FUNCTION_BLOCK FB_StringLookupElementMock EXTENDS FB_FalliblePublicMock IMPLEMENTS I_StringLookupElement;
VAR
    fAtomicMass : LREAL;
    nAtomicNumber : INT;
    fDensity : LREAL;
END_VAR

PROPERTY AtomicMass : LREAL
GET

AtomicMass := fAtomicMass;
END_GET
SET

fAtomicMass := AtomicMass;
END_SET
END_PROPERTY

PROPERTY AtomicNumber : INT
GET

AtomicNumber := nAtomicNumber;
END_GET
SET

nAtomicNumber := AtomicNumber;
END_SET
END_PROPERTY

PROPERTY Density : LREAL
GET

Density := fDensity;
END_GET
SET

fDensity := Density;
END_SET
END_PROPERTY


METHOD LookupAtomicMass : LREAL
VAR_INPUT
    sLookup	: STRING;
END_VAR

LookupAtomicMass := fAtomicMass;
END_METHOD


METHOD LookupAtomicNumber : INT
VAR_INPUT
    sLookup	: STRING;
END_VAR

LookupAtomicNumber := nAtomicNumber;
END_METHOD


METHOD LookupDensity : LREAL
VAR_INPUT
    sLookup	: STRING;
END_VAR

LookupDensity := fDensity;
END_METHOD


METHOD SetValid

fAtomicMass := 1.0;
nAtomicNumber := 1;
fDensity := 1.0;
END_METHOD

END_FUNCTION_BLOCK

(* stored: Version 1.1.0.1
   POU FB_StringLookupElementMock: Id {18e1cb23-bba9-4318-ba60-0ac68051a2a0}, SpecialFunc None
   Property AtomicMass: Id {635032a6-311e-4d7c-9b55-f9024148140d}
   Get Get: Id {f7c57037-db88-45ae-a7df-97c3b6733e71}
   Set Set: Id {6e4e3849-a0c8-41a4-8ebe-a5f025f04260}
   Property AtomicNumber: Id {06122f6b-f517-481a-9749-dc246c897461}
   Get Get: Id {e9d734fe-c826-493a-b424-586d3f706478}
   Set Set: Id {2b4c4e29-c09c-46cb-98bb-b25e81a01b1b}
   Property Density: Id {b79e1095-9dde-44a0-a231-d917464f7a3d}
   Get Get: Id {f0b638fa-d258-48cb-b13e-0dd7005455a7}
   Set Set: Id {8ff93d78-1bb5-4ac0-b979-6e67459ed291}
   Method LookupAtomicMass: Id {1dcfeecf-8505-43bc-a7d2-9b5fa59ddc2b}
   Method LookupAtomicNumber: Id {69859d7c-928a-4813-9e19-d45971dbc25d}
   Method LookupDensity: Id {c68ca04a-b56a-4ca8-ad9e-4621f979c04d}
   Method SetValid: Id {f7ff3f37-db96-476e-86c7-5553fd9ef068} *)
